INTERFACE itfCommand

METHOD Abort : MC_Error
VAR_INPUT
END_VAR
END_METHOD

PROPERTY Active : BOOL
GET
END_GET
SET
END_SET
END_PROPERTY

PROPERTY Busy : BOOL
GET
END_GET
SET
END_SET
END_PROPERTY

PROPERTY Command : MC_COMMAND_REF
GET
END_GET
SET
END_SET
END_PROPERTY

PROPERTY CommandAborted : BOOL
GET
END_GET
SET
END_SET
END_PROPERTY

PROPERTY Done : BOOL
GET
END_GET
SET
END_SET
END_PROPERTY

PROPERTY Error : BOOL
GET
END_GET
SET
END_SET
END_PROPERTY

PROPERTY ErrorId : MC_Error
GET
END_GET
SET
END_SET
END_PROPERTY

PROPERTY ErrorID_Udint : MC_ErrorID_Udint
GET
END_GET
SET
END_SET
END_PROPERTY

PROPERTY Status : BOOL
GET
END_GET
SET
END_SET
END_PROPERTY

METHOD Wait 		: MC_Error // This method only makes sense in the IEC 61499 environment
VAR_INPUT
	Timeout		 	: TIME;
	AbortOnTimeout 	: BOOL; 
END_VAR
END_METHOD

END_INTERFACE

(* stored: Version 1.1.0.1, ProductVersion 3.1.4024.12
   Itf itfCommand: Id {761ffb8a-079d-422c-ac48-277d623a645e}
   Method Abort: Id {44066283-c781-4c5d-9137-f7b260bddd39}
   Property Active: Id {49e914cc-c3e2-4cbb-9546-5b76536356ef}
   Get Get: Id {0ce9ab6e-faee-4368-8c97-873a6dbaae1f}
   Set Set: Id {63adf4f9-29e4-48a7-b498-da7a50a8fa33}
   Property Busy: Id {07bd0b04-ae26-4b1c-9339-e87c94820a63}
   Get Get: Id {1b11f855-47c2-4294-82c0-b75517bd4d8a}
   Set Set: Id {4f8a8617-1f5f-4b8f-b7db-8cc38454f89b}
   Property Command: Id {613ed526-2fc5-4bcf-8f97-8b8dba8f3f5c}
   Get Get: Id {eef50f13-0f9a-4e3e-a7ed-af5e33b9d6f1}
   Set Set: Id {b1d87a9c-5718-4563-95aa-e404be989a01}
   Property CommandAborted: Id {8b585279-c8af-4948-b7e6-a73c5ba6d655}
   Get Get: Id {085598aa-9a22-4404-9a68-c23969695b20}
   Set Set: Id {d07d5132-2041-4a7d-88cd-028e2b106d35}
   Property Done: Id {32454eeb-aaaa-4ab0-b761-d85aed51d1f7}
   Get Get: Id {ca9a4bf6-4742-4414-ac68-0b34bcf01142}
   Set Set: Id {2cc75574-2468-418b-bf11-553f5c967ded}
   Property Error: Id {bbbb4768-0975-443f-84fa-70b2255faee1}
   Get Get: Id {cf511c99-7bc4-44e2-9840-4e56131a64c0}
   Set Set: Id {b349f36a-4e77-4c97-b4d2-c08410b2b5fb}
   Property ErrorId: Id {20e7a598-13f3-4619-aa13-feb95d88f789}
   Get Get: Id {602d2ea6-902d-4220-abad-8c8f61e6666d}
   Set Set: Id {438d217c-a6b9-4581-aaad-a9b1c0dd7f00}
   Property ErrorID_Udint: Id {e9103c94-daac-4dc0-a702-4eec4267d376}
   Get Get: Id {49171e37-7f88-4b76-88ef-706332e921aa}
   Set Set: Id {f0327e1e-73b9-42df-819a-10d5a22dc523}
   Property Status: Id {49a8fca0-076d-4700-9b48-3b8c7dc690a4}
   Get Get: Id {028dfcb1-b6f5-4f46-afb1-561684af3ad7}
   Set Set: Id {6be722dd-a01d-414b-805c-a8b448b2e901}
   Method Wait: Id {6d8924ab-9a65-4615-99c1-0f1843870fe1} *)
